{attribute 'qualified_only'}
//{attribute 'strict'}
{attribute 'to_string'}
TYPE E_MESSAGE_STATE :
(
	MSG_STATE_NULL,
  MSG_STATE_INIT    := 10,
  MSG_STATE_IDLE    := 30,
  MSG_STATE_WRITE   := 50
)UINT;
END_TYPE

(* stored: Version 1.1.0.1
   DUT E_MESSAGE_STATE: Id {29f3033f-ad50-47d6-a1ef-1e06e7dbbcdb} *)
